VAR_GLOBAL
	{attribute 'OPC.UA.DA' := '1'}
	{attribute 'OPC.UA.DA.StructuredType' := '1'}
	{attribute 'OPC.UA.DA.Description' := 'Complex (structured) type '} 	
	StructuredType1 : ST_Complex_1;
	
	{attribute 'OPC.UA.DA' := '2'}
	{attribute 'OPC.UA.DA.StructuredType' := '1'}
	{attribute 'OPC.UA.DA.Description' := 'Complex (structured) type '} 	
	StructuredType1WithoutMember : ST_Complex_1;

	{attribute 'OPC.UA.DA' := '1'}
	{attribute 'OPC.UA.DA.StructuredType' := '1'}
	{attribute 'OPC.UA.DA.Description' := 'Complex (structured) type '} 		
	StructuredType2 : ST_Complex_2;
	
	{attribute 'OPC.UA.DA' := '1'}
	{attribute 'OPC.UA.DA.StructuredType' := '1'}
	{attribute 'OPC.UA.DA.Description' := 'Complex (structured) type '} 		
	StructuredType3 : ST_Complex_3;

	{attribute 'OPC.UA.DA' := '1'}
	{attribute 'OPC.UA.DA.StructuredType' := '1'}
	{attribute 'OPC.UA.DA.Description' := 'Complex (structured) type '} 		
	StructuredType4 : ST_Complex_4;	
	
	{attribute 'OPC.UA.DA' := '1'}
	{attribute 'OPC.UA.DA.StructuredType' := '1'}
	{attribute 'OPC.UA.DA.Description' := 'Complex (structured) type '} 		
	StructuredType5 : ST_Complex_5;	
	
	{attribute 'OPC.UA.DA' := '1'}
	{attribute 'OPC.UA.DA.StructuredType' := '1'}
	{attribute 'OPC.UA.DA.Description' := 'Complex (structured) type '} 		
	StructuredType6 : ST_Complex_6;	
	
	{attribute 'OPC.UA.DA' := '1'}
	{attribute 'OPC.UA.DA.StructuredType' := '1'}
	{attribute 'OPC.UA.DA.Description' := 'Complex (structured) type '} 		
	StructuredType7 : ST_Complex_7;		

	{attribute 'OPC.UA.DA' := '1'}
	{attribute 'OPC.UA.DA.StructuredType' := '1'}
	{attribute 'OPC.UA.DA.Description' := 'Complex (structured) type '} 		
	StructuredType8 : ST_Complex_8;	
	
	{attribute 'OPC.UA.DA' := '1'}
	{attribute 'OPC.UA.DA.StructuredType' := '1'}
	{attribute 'OPC.UA.DA.Description' := 'Array of complex (structured) type'} 	
	arrStComplex : ARRAY[0..ARRSIZEX] OF ST_Complex_1;

	{attribute 'OPC.UA.DA' := '1'}
	{attribute 'OPC.UA.DA.StructuredType' := '1'}
	{attribute 'OPC.UA.DA.Description' := 'Array of complex (structured) type'} 		
	arrStComplex2 : ARRAY[0..ARRSIZEX] OF ST_Complex_2;		
END_VAR

(* stored: Version 1.1.0.1
   GVL GVL_structures: Id {55b4d72c-7100-4385-be79-aa7caa1663d1} *)
